TYPE TelemetryAccelerometersStatuses :
STRUCT
	///Are all accelerometers in a healthy state?
	healthStatus: HealthStatus;
END_STRUCT
END_TYPE

(* stored: Version 1.1.0.1, ProductVersion 3.1.4019.2
   DUT TelemetryAccelerometersStatuses: Id {87e7d2c9-7991-4b04-9aab-98a94c7460d7} *)
